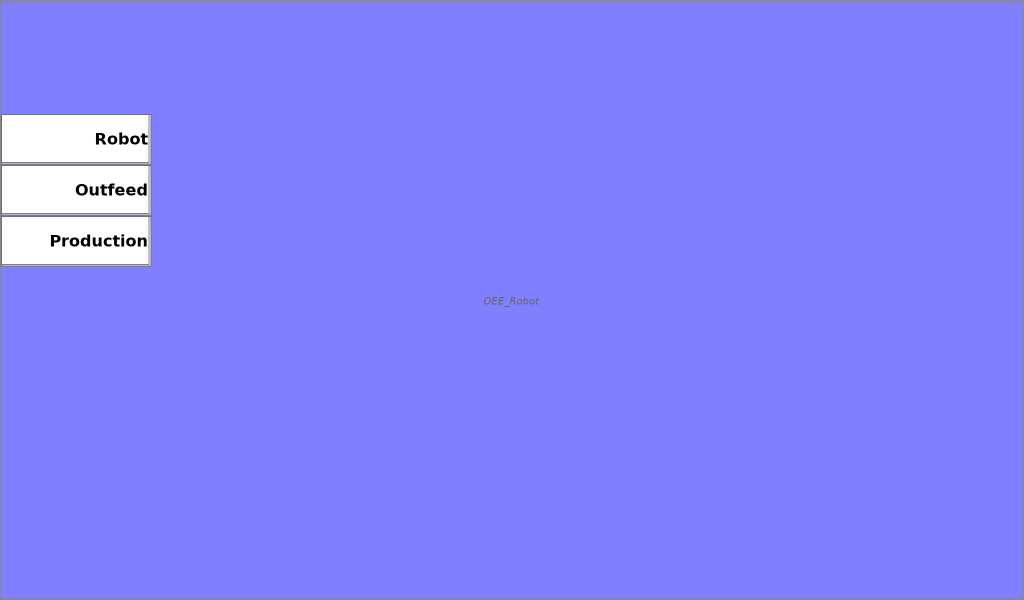
VISUALIZATION OEE  // 1024x600
    Frame (0,2 1023x598)
        shows OEE_Robot()
        shows OEE_Outfeed()
        shows OEE_Counter()
        shows Test_Place1()
        shows Test_Place2()
        shows Test_Place3()
        shows Test_Place4()
    Button (1,114 150x50), "Robot", image: VisuSymbols.Symbols.Database2
        OnMouseDown: FrameSelectionChange Selection=SelectedFrame=146e207b-fd78-4676-ba16-384fa245d7d2, GlobSel=AssignDir=MainPage.GenElemInst_1003, AssignType=Directly, SelType=Locally
    Button (1,165 150x50), "Outfeed", image: VisuSymbols.Symbols.Database2
        OnMouseDown: FrameSelectionChange Selection=SelectedFrame=146e207b-fd78-4676-ba16-384fa245d7d2, Selection=1, GlobSel=AssignDir=MainPage.GenElemInst_1003, AssignType=Directly, SelType=Locally
    Button (1,216 150x50), "Production", image: VisuSymbols.Symbols.Database2
        OnMouseDown: FrameSelectionChange Selection=SelectedFrame=146e207b-fd78-4676-ba16-384fa245d7d2, Selection=2, GlobSel=AssignDir=MainPage.GenElemInst_1003, AssignType=Directly, SelType=Locally
END_VISUALIZATION

(* stored: Version 1.1.0.1, ProductVersion 3.1.4024.12
   Visu OEE: Id {6bf23cef-9e7d-4b81-a9c7-2e2cf4132284} *)
